TYPE ST_INPUTS_DrumFilter:
STRUCT
	
	Mode:     		E_DeviceMode;
	Command:     E_DeviceState;

END_STRUCT
END_TYPE

(* stored: Version 1.1.0.1, ProductVersion 3.1.4024.12
   DUT ST_INPUTS_DrumFilter: Id {663cca9d-47ec-4333-a59e-0b26a15a1436} *)
